{attribute 'qualified_only'}
VAR_GLOBAL	
	extrusionWeight : REAL;
	
	extrusionHeight : REAL;
	extrusionWidth : REAL;
END_VAR

(* stored: Version 1.1.0.1, ProductVersion 3.1.4024.11
   GVL ExtrusionData: Id {16305a3b-4d45-4e59-8191-641eeb16f61f} *)
